(* Logix 5000 project; controller OPC_SAMPLE vendor 1 type 14 code 94 rev 19.53; software revision 19.01 *)

TASK MainTask (continuous, watchdog 500 ms) : MainProgram

MODULES
   Local : vendor 1 type 14 code 94 (ICP 0, rev 19.53)
END_MODULES

PROGRAM MainProgram   (* main routine MainRoutine *)
VAR
   INPUT : BOOL := 1;
   OUTPUT1 : BOOL := 1;
   OUTPUT2 : BOOL := 1;
   TIMER1 : TIMER := (PRE := 1000, ACC := 1000, EN := 1, DN := 1);
   TIMER2 : TIMER := (PRE := 1000, ACC := 389, EN := 1, TT := 1);
END_VAR

ROUTINE MainRoutine   (* ladder *)
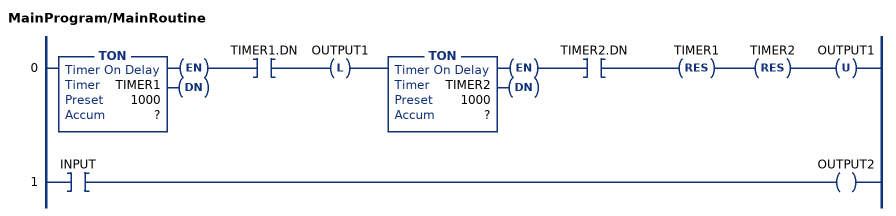
   0: TON(TIMER1,?,?)XIC(TIMER1.DN)OTL(OUTPUT1)TON(TIMER2,?,?)XIC(TIMER2.DN)RES(TIMER1)RES(TIMER2)OTU(OUTPUT1);
   1: XIC(INPUT)OTE(OUTPUT2);
END_ROUTINE
END_PROGRAM
